// TIA Portal V16 export
// export: Created 2024-12-03T15:41:44.5228332Z, ExportSetting WithDefaults, DisplayName Totally Integrated Automation Portal, DisplayVersion V16 Update 6, DisplayName TIA Portal Version Control Interface, DisplayVersion V16 Update 2, DisplayName TIA Portal Openness, DisplayVersion V16 Update 6, DisplayName TIA Portal Teamcenter Gateway, DisplayVersion V16, DisplayName SINAMICS Startdrive Advanced, DisplayVersion V16 Update 5, DisplayName SINAMICS Startdrive G130, G150, S120, S150, SINAMICS MV, S210, DisplayVersion V16 Update 5, DisplayName SINAMICS Startdrive G110M, G120, G120C, G120D, G120P, G115D, DisplayVersion V16 Update 5, DisplayName STEP 7 Professional, DisplayVersion V16 Update 6, DisplayName STEP 7 Safety, DisplayVersion V16, DisplayName WinCC Advanced / Unified PC, DisplayVersion V16 Update 6
DATA_BLOCK "EMG_STATUS_DB"   // DB85
{ S7_Optimized_Access := 'FALSE' }
VERSION : 0.1
// stored: AutoNumber true, DBAccessibleFromOPCUA true, IsOnlyStoredInLoadMemory false, IsWriteProtectedInAS false
   VAR
      EMG_MAIN : "EMG_Status_UDT";
      EMG_ZONE_1 : "EMG_Status_UDT";
      EMG_ZONE_2 : "EMG_Status_UDT";
      EMG_ZONE_3_4 { S7_SetPoint := 'True'} : "EMG_Status_UDT";
      EMG_ZONE_5 { S7_SetPoint := 'True'} : "EMG_Status_UDT";
   END_VAR
BEGIN
END_DATA_BLOCK
